// TIA Portal V17 export
// export: Created 2024-08-20T13:26:11.6505374Z, ExportSetting WithDefaults, DisplayName Totally Integrated Automation Portal, DisplayVersion V17 Update 4, DisplayName TIA Portal Openness, DisplayVersion V17 Update 4, DisplayName TIA Portal Version Control Interface, DisplayVersion V17, DisplayName STEP 7 Professional, DisplayVersion V17 Update 4, DisplayName STEP 7 Safety, DisplayVersion V17, DisplayName WinCC Advanced, DisplayVersion V17 Update 4
DATA_BLOCK "ROD4_DB"   // DB9
VERSION : 0.1
// stored: AutoNumber true, DBAccessibleFromOPCUA true, InstanceOfName ROD4, InstanceOfType FB
"ROD4"
   // VAR_INPUT
   //    G1OK : Bool;
   //    G2OK : Bool;
   //    G3OK : Bool;
   //    G4OK : Bool;
   //    G1L : Bool;
   //    G2L : Bool;
   //    G3L : Bool;
   //    G4L : Bool;
   //    TEROD : DInt;
   //    LIGP : Bool;
   //    LIGC1 : Bool;
   //    LIGC2 : Bool;
   //    LIGC3 : Bool;
   //    DESAB : Bool;
   //    T1S : Bool;
   // END_VAR
   // VAR_OUTPUT
   //    G1P : Bool;
   //    G2P : Bool;
   //    G3P : Bool;
   //    G4P : Bool;
   //    G1C1 : Bool;
   //    G2C1 : Bool;
   //    G3C1 : Bool;
   //    G4C1 : Bool;
   //    G1C2 : Bool;
   //    G2C2 : Bool;
   //    G3C2 : Bool;
   //    G4C2 : Bool;
   //    G1C3 : Bool;
   //    G2C3 : Bool;
   //    G3C3 : Bool;
   //    G4C3 : Bool;
   //    LG1 : Bool;
   //    LG2 : Bool;
   //    LG3 : Bool;
   //    LG4 : Bool;
   // END_VAR
   // VAR_IN_OUT
   //    TOG1P : DInt;
   //    TOG2P : DInt;
   //    TOG3P : DInt;
   //    TOG4P : DInt;
   //    TEOKG1 : Real;
   //    TEOKG2 : Real;
   //    TEOKG3 : Real;
   //    TEOKG4 : Real;
   // END_VAR
   // VAR
   //    GR1SELP : Bool;
   //    GR2SELP : Bool;
   //    GR3SELP : Bool;
   //    GR4SELP : Bool;
   //    GR1SELC1 : Bool;
   //    GR2SELC1 : Bool;
   //    GR3SELC1 : Bool;
   //    GR4SELC1 : Bool;
   //    GR1SELC2 : Bool;
   //    GR2SELC2 : Bool;
   //    GR3SELC2 : Bool;
   //    GR4SELC2 : Bool;
   //    GR1SELC3 : Bool;
   //    GR2SELC3 : Bool;
   //    GR3SELC3 : Bool;
   //    GR4SELC3 : Bool;
   //    PS1SG1 : Bool;
   //    PS1SG2 : Bool;
   //    PS1SG3 : Bool;
   //    PS1SG4 : Bool;
   //    PS1 : Bool;
   //    PS2 : Bool;
   //    PS3 : Bool;
   //    PS4 : Bool;
   //    FIMTEG1 : Bool;
   //    FIMTEG2 : Bool;
   //    FIMTEG3 : Bool;
   //    FIMTEG4 : Bool;
   //    SDESG1 : Bool;
   //    SDESG2 : Bool;
   //    SDESG3 : Bool;
   //    SDESG4 : Bool;
   //    GPL : Bool;
   //    GC1L : Bool;
   //    GC2L : Bool;
   //    GC3L : Bool;
   //    SO_L : Bool;
   //    SO_D : Bool;
   //    RTEOKG1 : Bool;
   //    RTEOKG2 : Bool;
   //    RTEOKG3 : Bool;
   //    RTEOKG4 : Bool;
   //    TON1 { S7_SetPoint := 'True'} : TON_TIME;
   //    TON2 { S7_SetPoint := 'True'} : TON_TIME;
   //    TON3 { S7_SetPoint := 'True'} : TON_TIME;
   //    TON4 { S7_SetPoint := 'True'} : TON_TIME;
   //    TSDG1 { S7_SetPoint := 'True'} : TON_TIME;
   //    TSDG2 { S7_SetPoint := 'True'} : TON_TIME;
   //    TSDG3 { S7_SetPoint := 'True'} : TON_TIME;
   //    TSDG4 { S7_SetPoint := 'True'} : TON_TIME;
   // END_VAR
BEGIN
END_DATA_BLOCK
